SUBAPPLICATION Uebung_086_AX (* Beispiel für E_SWITCH, mit Plug and Socket *)
  (* Standard: 61499-2; Description: Copyright (c) 2026 Meisterschulen am Ostbahnhof This program and the accompanying materials are made available under the terms of the Eclipse Public License 2.0 which is available at https://www.eclipse.org/legal/epl-2.0/ SPDX-License-Identifier: EPL-2.0 *)
  (* Version 1.0, 2026-09-10, Franz Höpfinger, Meisterschulen am Ostbahnhof, initial API and implementation and/or initial documentation *)
  PACKAGE Uebungen;
  IMPORT logiBUS::io::DI::logiBUS_DI::Input_I1;
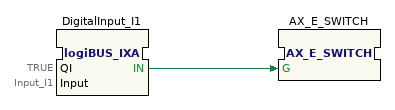
  FBS
    DigitalInput_I1 : logiBUS::io::DI::logiBUS_IXA(QI := TRUE, Input := Input_I1);
    AX_E_SWITCH : adapter::events::unidirectional::AX_E_SWITCH;
  END_FBS
  ADAPTER_CONNECTIONS
    DigitalInput_I1.IN TO AX_E_SWITCH.G;
  END_CONNECTIONS
END_SUBAPPLICATION
